SYSTEM FbeTestProject
  (* Standard: Test standard; Classification: Test; ApplicationDomain: GASR; Function: For testing; Type: Test; Description: System created for test purposes only *)
  (* Version 1.0, 2024-05-15, cabral, GASR-UDESC *)
  APPLICATION MainApp
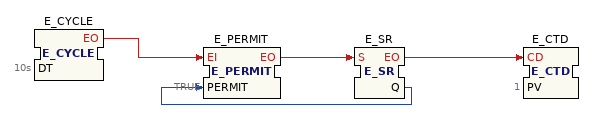
    FBS
      E_SR : E_SR;
      E_PERMIT : E_PERMIT(PERMIT := TRUE);
      E_CYCLE : E_CYCLE(DT := 10s);
      E_CTD : E_CTD(PV := 1);
    END_FBS
    EVENT_CONNECTIONS
      E_CYCLE.EO TO E_PERMIT.EI;
      E_PERMIT.EO TO E_SR.S;
      E_SR.EO TO E_CTD.CD;
    END_CONNECTIONS
    DATA_CONNECTIONS
      E_SR.Q TO E_PERMIT.PERMIT;
    END_CONNECTIONS
  END_APPLICATION
  APPLICATION SumApp
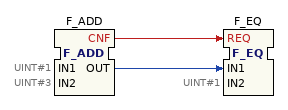
    FBS
      F_ADD : F_ADD(IN1 := UINT#1, IN2 := UINT#3);
      F_EQ : F_EQ(IN2 := UINT#1);
    END_FBS
    EVENT_CONNECTIONS
      F_ADD.CNF TO F_EQ.REQ;
    END_CONNECTIONS
    DATA_CONNECTIONS
      F_ADD.OUT TO F_EQ.IN1;
    END_CONNECTIONS
  END_APPLICATION
  APPLICATION MultApp
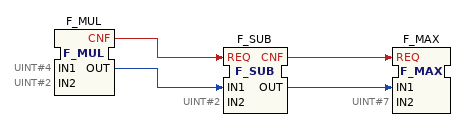
    FBS
      F_MUL : F_MUL(IN1 := UINT#4, IN2 := UINT#2);
      F_SUB : F_SUB(IN2 := UINT#2);
      F_MAX : F_MAX(IN2 := UINT#7);
    END_FBS
    EVENT_CONNECTIONS
      F_MUL.CNF TO F_SUB.REQ;
      F_SUB.CNF TO F_MAX.REQ;
    END_CONNECTIONS
    DATA_CONNECTIONS
      F_MUL.OUT TO F_SUB.IN1;
      F_SUB.OUT TO F_MAX.IN1;
    END_CONNECTIONS
  END_APPLICATION
  DEVICE DEV_FORTE : FORTE_PC(MGR_ID := "localhost:61499")
    {SET_ATTRIBUTE(Profile, HOLOBLOC)} (* device profile *)
    RESOURCE FST_RES : EMB_RES
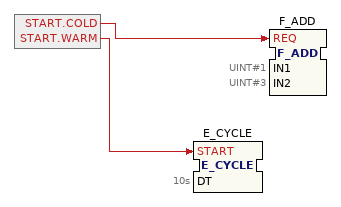
      FBS
        F_ADD : F_ADD(IN1 := UINT#1, IN2 := UINT#3);
        E_CYCLE : E_CYCLE(DT := 10s);
      END_FBS
      EVENT_CONNECTIONS
        START.COLD TO F_ADD.REQ;
        START.WARM TO E_CYCLE.START;
      END_CONNECTIONS
    END_RESOURCE
    RESOURCE SECOND_RES : EMB_RES
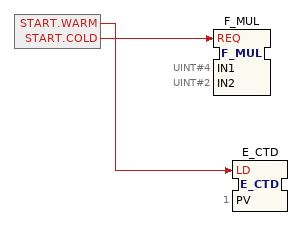
      FBS
        E_CTD : E_CTD(PV := 1);
        F_MUL : F_MUL(IN1 := UINT#4, IN2 := UINT#2);
      END_FBS
      EVENT_CONNECTIONS
        START.WARM TO E_CTD.LD;
        START.COLD TO F_MUL.REQ;
      END_CONNECTIONS
    END_RESOURCE
    RESOURCE THIRD_RES : EMB_RES
    END_RESOURCE
  END_DEVICE
  DEVICE FORTE : FORTE_PC(MGR_ID := "localhost:61499")
    {SET_ATTRIBUTE(Profile, HOLOBLOC)} (* device profile *)
    RESOURCE GASR : EMB_RES
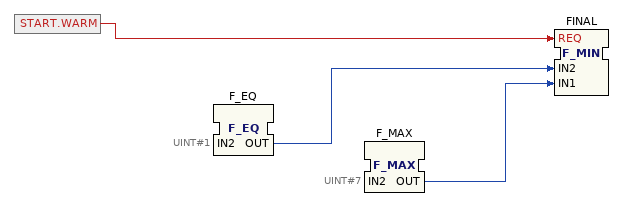
      FBS
        F_EQ : F_EQ(IN2 := UINT#1);
        FINAL : F_MIN;
        F_MAX : F_MAX(IN2 := UINT#7);
      END_FBS
      EVENT_CONNECTIONS
        START.WARM TO FINAL.REQ;
      END_CONNECTIONS
      DATA_CONNECTIONS
        F_EQ.OUT TO FINAL.IN2;
        F_MAX.OUT TO FINAL.IN1;
      END_CONNECTIONS
    END_RESOURCE
  END_DEVICE
  MAPPINGS
    SumApp.F_ADD ON DEV_FORTE.FST_RES.F_ADD;
    MainApp.E_CYCLE ON DEV_FORTE.FST_RES.E_CYCLE;
    MainApp.E_CTD ON DEV_FORTE.SECOND_RES.E_CTD;
    SumApp.F_EQ ON FORTE.GASR.F_EQ;
    MultApp.F_MAX ON FORTE.GASR.F_MAX;
    MultApp.F_MUL ON DEV_FORTE.SECOND_RES.F_MUL;
  END_MAPPINGS
END_SYSTEM
